// TwinCAT 3 PLC project ProjectA
// ProgramVersion: 3.1.4022.7
// libraries:
//   Tc2_Standard, * (Beckhoff Automation GmbH)
//   Tc2_System, * (Beckhoff Automation GmbH)
//   Tc3_Module, * (Beckhoff Automation GmbH)
// project tree:
//   DUTs/ ST_ProjectA.TcDUT
//   GVLs/ GVL_ProjectA.TcGVL, ParameterList.TcGVL
//   / PlcTask.TcTTO
//   POUs/ FB_ProjectA.TcPOU, MAIN.TcPOU
//   Unsupported/ ClassDiagram.TcCD (not stored), GlobalTextList.TcGTLO, ImagePool.TcIPO (not stored), RecipeManager.TcRMO (not stored), TextList.TcTLO
// real-time tasks:
//   TASK PlcTask: cycle T#10ms, priority 20, ADS port 350

CONFIGURATION ProjectA
    RESOURCE PLC ON TwinCAT3
        TASK PlcTask(INTERVAL := T#10ms, PRIORITY := 20);
        PROGRAM MAIN WITH PlcTask : MAIN;
    END_RESOURCE
END_CONFIGURATION

// ---- DUTs/ST_ProjectA.TcDUT
TYPE ST_ProjectA :
STRUCT
	iValue : INT;
END_STRUCT
END_TYPE

// ---- GVLs/GVL_ProjectA.TcGVL
{attribute 'qualified_only'}
VAR_GLOBAL
	bProjectA : BOOL := FALSE;
END_VAR

// ---- GVLs/ParameterList.TcGVL
{attribute 'qualified_only'}
VAR_GLOBAL CONSTANT
	iParamList : INT := 1;
END_VAR

// ---- POUs/MAIN.TcPOU
PROGRAM MAIN
VAR
END_VAR

END_PROGRAM

// ---- POUs/FB_ProjectA.TcPOU
FUNCTION_BLOCK FB_ProjectA
VAR_INPUT
	fValue : LREAL;
END_VAR
VAR_OUTPUT
END_VAR
VAR
END_VAR

fValue := 1.0;

END_FUNCTION_BLOCK

// ---- Unsupported/TextList.TcTLO
TEXTLIST TextList
   = ''
END_TEXTLIST
